(* CODESYS project Prova_Ladder_and_ST.project

Project tree, tasks and I/O mapping:
  Device : CODESYS Control Win V3, 3S - Smart Software Solutions GmbH, order no. 305021, version 3.5.10.30
    application Application
      libraries: Standard, * (System)
      task MainTask (cyclic, interval t#20ms, priority 1) calls PLC_PRG, ST_PRG
      task VISU_TASK (cyclic, interval 100 ms, priority 31) calls VisuElems.Visu_Prg
      program PLC_PRG [LD]
      visualisation Visualization
      program ST_PRG [ST]
  text list GlobalTextList
*)

// Device/Application/PLC_PRG
PROGRAM PLC_PRG
VAR
	Contact1: BOOL := FALSE;
	Coil1: BOOL := FALSE;
END_VAR

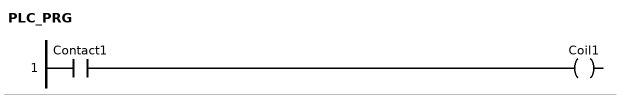
// NETWORK 1
Coil1 := Contact1;

END_PROGRAM

// Device/Application/ST_PRG
PROGRAM ST_PRG
VAR
	Contact1 : BOOL := FALSE;
	Coil1 : BOOL := FALSE;
END_VAR

Coil1 := Contact1;

(* PLC_PRG.Coil1 := PLC_PRG.Contact1; *)

END_PROGRAM

// Device/Application/Visualization
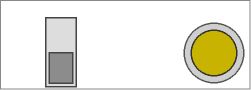
VISUALIZATION Visualization  // 251x90
    DipSwitch (26,17 70x70), variable: PLC_PRG.Contact1, behaviour: TOGGLE, style: Switch-DipSwitch-Gray
    Lamp1 (179,18 70x70), variable: PLC_PRG.Coil1, style: Lamp-Lamp1-Yellow
END_VISUALIZATION
